SUBAPPLICATION VT_active (* Subapplication Type *)
  (* Standard: 61499-2 *)
  (* Version 1.0, 2023-02-19, franz *)
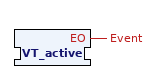
  EVENT_OUTPUT
    EO;
  END_EVENT
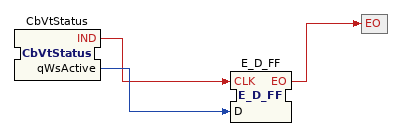
  FBS
    E_D_FF : E_D_FF;
    CbVtStatus : CbVtStatus;
  END_FBS
  EVENT_CONNECTIONS
    E_D_FF.EO TO EO;
    CbVtStatus.IND TO E_D_FF.CLK;
  END_CONNECTIONS
  DATA_CONNECTIONS
    CbVtStatus.qWsActive TO E_D_FF.D;
  END_CONNECTIONS
END_SUBAPPLICATION
